FUNCTION_BLOCK SFC2_SFC3_VIEW (* Composite Function Block Type *)
  (* Standard: 61499-2 *)
  (* Version 0.2, 2003-12-05, JHC, Rockwell Automation, Renamed from NEWCOMPFB. *)
  (* Version 0.1, 2002-01-08, JHC, Rockwell Automation, Added DLY FB as example. *)
  (* Version 0.0, 2000-05-27, JHC, Rockwell Automation *)
  (* Compiler header: package fb.rt.pnp;import fb.rt.vhmi.*; *)
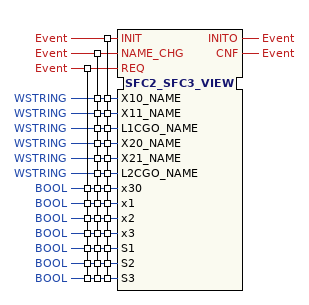
  EVENT_INPUT
    INIT WITH X10_NAME, X11_NAME, L1CGO_NAME, X20_NAME, X21_NAME, L2CGO_NAME, x30, x1, S1, x3, S3, x2, S2; (* Initialization Request *)
    NAME_CHG WITH X10_NAME, X11_NAME, L1CGO_NAME, X20_NAME, X21_NAME, L2CGO_NAME, x30, x1, S1, x3, S3, x2, S2; (* Normal Execution Request *)
    REQ WITH x30, x1, S1, x3, S3, x2, S2;
  END_EVENT
  EVENT_OUTPUT
    INITO; (* Initialization Confirm *)
    CNF; (* Execution Confirmation *)
  END_EVENT
  VAR_INPUT
    X10_NAME : WSTRING; (* Input event qualifier *)
    X11_NAME : WSTRING;
    L1CGO_NAME : WSTRING;
    X20_NAME : WSTRING;
    X21_NAME : WSTRING;
    L2CGO_NAME : WSTRING;
    x30 : BOOL;
    x1 : BOOL;
    x2 : BOOL;
    x3 : BOOL;
    S1 : BOOL;
    S2 : BOOL;
    S3 : BOOL;
  END_VAR
  FBS
    X10 : Render(Display := 1, Layer := 2, PosX := 105, PosY := 305);
    X11 : Render(Display := 1, Layer := 2, PosX := 105, PosY := 374);
    L1CGO : Render(Display := 1, Layer := 2, PosX := 179, PosY := 375);
    SFC3 : Render(name := "/fb/rt/pnp/pics/SFC3.png", PosX := 25, PosY := 453, Display := 1, Layer := 1);
    X20 : Render(Display := 1, Layer := 2, PosX := 105, PosY := 508);
    X21 : Render(Display := 1, Layer := 2, PosX := 105, PosY := 577);
    L2CGO : Render(Display := 1, Layer := 2, PosX := 179, PosY := 578);
    SFC2 : Render(name := "/fb/rt/pnp/pics/SFC2.png", PosX := 25, PosY := 250, Display := 1, Layer := 1);
    X30 : Render(name := "/fb/rt/pnp/pics/DASH.png", Layer := 2, PosX := 163, PosY := 366);
    X1 : Render(name := "/fb/rt/pnp/pics/DASH.png", Layer := 2, PosY := 366, PosX := 193);
    Ns1 : Render(name := "/fb/rt/pnp/pics/DASH.png", Layer := 2, PosX := 213, PosY := 366);
    X3 : Render(name := "/fb/rt/pnp/pics/DASH.png", Layer := 2, PosX := 240, PosY := 366);
    Ns3 : Render(name := "/fb/rt/pnp/pics/DASH.png", Layer := 2, PosX := 259, PosY := 366);
    X1_1 : Render(name := "/fb/rt/pnp/pics/DASH.png", Layer := 2, PosY := 445, PosX := 157);
    s1 : Render(name := "/fb/rt/pnp/pics/DASH.png", Layer := 2, PosY := 445, PosX := 177);
    X3_1 : Render(name := "/fb/rt/pnp/pics/DASH.png", Layer := 2, PosY := 445, PosX := 203);
    s3 : Render(name := "/fb/rt/pnp/pics/DASH.png", Layer := 2, PosY := 445, PosX := 223);
    NotS1 : NotGate;
    NotS3 : NotGate;
    X30_1 : Render(name := "/fb/rt/pnp/pics/DASH.png", Layer := 2, PosX := 162, PosY := 570);
    X2 : Render(name := "/fb/rt/pnp/pics/DASH.png", Layer := 2, PosY := 570, PosX := 194);
    Ns2 : Render(name := "/fb/rt/pnp/pics/DASH.png", Layer := 2, PosY := 570, PosX := 213);
    X3_2 : Render(name := "/fb/rt/pnp/pics/DASH.png", Layer := 2, PosY := 570, PosX := 239);
    Ns3_1 : Render(name := "/fb/rt/pnp/pics/DASH.png", Layer := 2, PosY := 570, PosX := 259);
    X2_1 : Render(name := "/fb/rt/pnp/pics/DASH.png", Layer := 2, PosY := 648, PosX := 157);
    s2_1 : Render(name := "/fb/rt/pnp/pics/DASH.png", Layer := 2, PosY := 648, PosX := 177);
    X3_3 : Render(name := "/fb/rt/pnp/pics/DASH.png", Layer := 2, PosY := 648, PosX := 203);
    s3_1 : Render(name := "/fb/rt/pnp/pics/DASH.png", Layer := 2, PosY := 648, PosX := 223);
    NS2Gate : NotGate;
  END_FBS
  EVENT_CONNECTIONS
    INIT TO SFC2.INIT;
    SFC2.INITO TO X10.INIT;
    X10.INITO TO X11.INIT;
    X11.INITO TO L1CGO.INIT;
    X20.INITO TO X21.INIT;
    X21.INITO TO L2CGO.INIT;
    X10.CNF TO X11.ChangePic;
    X11.CNF TO L1CGO.ChangePic;
    X20.CNF TO X21.ChangePic;
    X21.CNF TO L2CGO.ChangePic;
    L2CGO.INITO TO X30.INIT;
    X30.INITO TO X1.INIT;
    Ns1.INITO TO X3.INIT;
    Ns3.INITO TO X1_1.INIT;
    X1_1.INITO TO s1.INIT;
    s1.INITO TO X3_1.INIT;
    X3_1.INITO TO s3.INIT;
    X30.CNF TO X1.ChangeValidity;
    Ns1.CNF TO X3.ChangeValidity;
    Ns3.CNF TO X1_1.ChangeValidity;
    X1_1.CNF TO s1.ChangeValidity;
    s1.CNF TO X3_1.ChangeValidity;
    X3_1.CNF TO s3.ChangeValidity;
    X1.INITO TO NotS1.INIT;
    NotS1.INITO TO Ns1.INIT;
    X1.CNF TO NotS1.REQ;
    NotS1.CNF TO Ns1.ChangeValidity;
    X3.INITO TO NotS3.INIT;
    NotS3.INITO TO Ns3.INIT;
    NotS3.CNF TO Ns3.ChangeValidity;
    X3.CNF TO NotS3.REQ;
    NAME_CHG TO X10.ChangePic;
    REQ TO X30.ChangeValidity;
    L1CGO.INITO TO SFC3.INIT;
    SFC3.INITO TO X20.INIT;
    L1CGO.CNF TO X20.ChangePic;
    s3.INITO TO X30_1.INIT;
    s3.CNF TO X30_1.ChangeValidity;
    X30_1.CNF TO X2.ChangeValidity;
    X30_1.INITO TO X2.INIT;
    Ns2.INITO TO X3_2.INIT;
    X3_2.INITO TO Ns3_1.INIT;
    Ns3_1.INITO TO X2_1.INIT;
    X2_1.INITO TO s2_1.INIT;
    s2_1.INITO TO X3_3.INIT;
    X3_3.INITO TO s3_1.INIT;
    Ns2.CNF TO X3_2.ChangeValidity;
    X3_2.CNF TO Ns3_1.ChangeValidity;
    Ns3_1.CNF TO X2_1.ChangeValidity;
    X2_1.CNF TO s2_1.ChangeValidity;
    s2_1.CNF TO X3_3.ChangeValidity;
    X3_3.CNF TO s3_1.ChangeValidity;
    s3_1.INITO TO INITO;
    s3_1.CNF TO CNF;
    X2.INITO TO NS2Gate.INIT;
    NS2Gate.INITO TO Ns2.INIT;
    X2.CNF TO NS2Gate.REQ;
    NS2Gate.CNF TO Ns2.ChangeValidity;
  END_CONNECTIONS
  DATA_CONNECTIONS
    X10_NAME TO X10.name;
    X11_NAME TO X11.name;
    L1CGO_NAME TO L1CGO.name;
    X20_NAME TO X20.name;
    X21_NAME TO X21.name;
    L2CGO_NAME TO L2CGO.name;
    x30 TO X30.Display;
    x1 TO X1.Display;
    x3 TO X3.Display;
    x1 TO X1_1.Display;
    S1 TO s1.Display;
    x3 TO X3_1.Display;
    S3 TO s3.Display;
    NotS1.QO TO Ns1.Display;
    S1 TO NotS1.QI;
    NotS3.QO TO Ns3.Display;
    S3 TO NotS3.QI;
    x30 TO X30_1.Display;
    x2 TO X2.Display;
    NS2Gate.QO TO Ns2.Display;
    S2 TO NS2Gate.QI;
    x3 TO X3_2.Display;
    NotS3.QO TO Ns3_1.Display;
    x2 TO X2_1.Display;
    S2 TO s2_1.Display;
    x3 TO X3_3.Display;
    S3 TO s3_1.Display;
  END_CONNECTIONS
END_FUNCTION_BLOCK
